Fanuc KAREL source: kb00021.KL

-- PROVISIONAL review KL for V1013-1; original PC SHA256 ba3e9bbd21b5904b23d3e01746366395855c0a2c136e3c2dfbf30341f36a7589
-- Incomplete behavior may be omitted. Consult companion uncertainty JSON. Do not deploy.
PROGRAM KB00021
%NOLOCKGROUP
BEGIN
  -- UNRESOLVED_PC offsets 5-14; opcodes 3F,75
  -- UNRESOLVED_PC offsets 19-26; opcodes 9D,23
  -- UNRESOLVED_PC offsets 31-49; opcodes 27,22,2A,22,31
  -- UNRESOLVED_PC offsets 54-58; opcodes 7F
END KB00021
